{attribute 'qualified_only'}
{attribute 'strict'}
TYPE E_StatesAteqRecipeHandler :
(
	RECIPE_IDLE,
	RECIPE_TRIGGER_VALVES, 	// From Mask
	RECIPE_WAIT_VALVES,		// Stabilization
	RECIPE_RUN_ATEQ,
	RECIPE_STORE_RESULTS,
	RECIPE_ERROR,
	RECIPE_TIMEOUT
);
END_TYPE

(* stored: Version 1.1.0.1, ProductVersion 3.1.4024.15
   DUT E_StatesAteqRecipeHandler: Id {1c794de3-b3b4-42f6-98c2-670725542067} *)
